// TIA Portal V20 export
TYPE "UDT_MTP_MonBinDrvSpd"
   STRUCT
      Spd1En : Bool;
      Spd2En : Bool;
      StopOp : Bool := FALSE;
      Spd1Op : Bool := FALSE;
      Spd2Op : Bool := FALSE;
      OSLevel : Byte := 16#00;
      StateChannel : Bool;
      StateOffAut : Bool;
      StateOffOp : Bool;
      StateOpAut : Bool;
      StateOpOp : Bool;
      StateAutAut : Bool;
      StateAutOp : Bool;
      StateOpAct : Bool;
      StateAutAct : Bool;
      StateOffAct : Bool;
      SafePos : Bool;
      CSF : Bool;
      WQC : Byte := 16#80;
      StopAut : Bool := FALSE;
      Spd1Aut : Bool := FALSE;
      Spd2Aut : Bool := FALSE;
      Spd1Ctrl : Bool := FALSE;
      Spd2Ctrl : Bool := FALSE;
      Spd2FbkCalc : Bool;
      Spd1FbkCalc : Bool;
      Spd2Fbk : Bool := FALSE;
      Spd1Fbk : Bool := FALSE;
      Trip : Bool := FALSE;
      PermEn : Bool := FALSE;
      Permit : Bool := FALSE;
      IntlEn : Bool := FALSE;
      Interlock : Bool := FALSE;
      ProtEn : Bool := FALSE;
      Protect : Bool := FALSE;
      ResetOp : Bool := FALSE;
      ResetAut : Bool := FALSE;
      MonEn : Bool := FALSE;
      MonSafePos : Bool := FALSE;
      MonStatErr : Bool := FALSE;
      MonDynErr : Bool := FALSE;
      MonStatTi : Real := 0.0;
      MonDynTi : Real := 0.0;
   END_STRUCT;
END_TYPE
